FUNCTION_BLOCK TAdsReadWrite
VAR_INPUT
END_VAR
VAR_OUTPUT
END_VAR
VAR
    AdsReadWrite : ADSRDWRT;
    Execution : TExecution;
END_VAR

AdsReadWrite(
	NETID:= , 
	PORT:= , 
	IDXGRP:= , 
	IDXOFFS:= , 
	WRITELEN:= , 
	READLEN:= , 
	SRCADDR:= , 
	DESTADDR:= , 
	WRTRD:= Execution.Starting, 
	TMOUT:= , 
	BUSY=> , 
	ERR=> , 
	ERRID=> );
    
IF Execution.Starting THEN
    Execution.SetBusy();
END_IF
IF Execution.Busy AND NOT AdsReadWrite.BUSY THEN
    IF AdsReadWrite.ERR THEN
        Execution.SetError(AdsReadWrite.ERRID);
    ELSE
        Execution.SetDone();
	END_IF
END_IF

METHOD Execute : BOOL
VAR_INPUT
    AmsNetId             : T_AmsNetID;
    Port                 : T_AmsPort;
    IndexGroup           : UDINT;
    IndexOffset          : UDINT; 
    ArgsAddress          : PVOID; 
    ArgsLength           : UDINT; 
    ReturnValueAddress   : PVOID; 
    ReturnValueLength    : UDINT; 
END_VAR
IF Execution.Start() THEN
    AdsReadWrite.NETID    := AmsNetId;
    AdsReadWrite.PORT     := Port;
    AdsReadWrite.IDXGRP   := IndexGroup;
    AdsReadWrite.IDXOFFS  := IndexOffset;
    // Data to be written...
    AdsReadWrite.SRCADDR  := ArgsAddress;
    AdsReadWrite.WRITELEN := ArgsLength;
    // Data returned...
    AdsReadWrite.DESTADDR := ReturnValueAddress;
    AdsReadWrite.READLEN  := ReturnValueLength;
END_IF
END_METHOD

PROPERTY ExecutionResult : IExecutionResult
GET
ExecutionResult := Execution;
END_GET
END_PROPERTY

END_FUNCTION_BLOCK

(* stored: Version 1.1.0.1, ProductVersion 3.1.4022.12
   POU TAdsReadWrite: Id {5aec252a-cd25-0680-3f48-2fefdad531b3}, SpecialFunc None
   Method Execute: Id {3b6f6d27-4076-0e86-0c12-92bfcd385060}
   Property ExecutionResult: Id {c61d60c8-81bd-0935-03bc-90d31f301497}
   Get Get: Id {00804ebf-72f7-0d30-3576-8dfddec5d3ed} *)
